FUNCTION_BLOCK UR (* Tamplate for a simple Basic Function Block Type *)
  (* Standard: 61499-2 *)
  (* Version 0.0, 2018-01-18, 4DIAC-IDE, 4DIAC-Consortium *)
  (* Version 1.0, 2016-05-26, AZ, fortiss GmbH *)
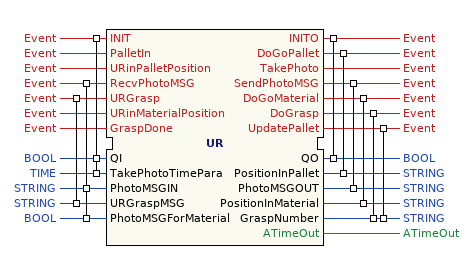
  EVENT_INPUT
    INIT WITH QI, TakePhotoTimePara; (* Initialization Request *)
    PalletIn; (* Normal Execution Request *)
    URinPalletPosition;
    RecvPhotoMSG WITH PhotoMSGIN, PhotoMSGForMaterial;
    URGrasp WITH URGraspMSG;
    URinMaterialPosition;
    GraspDone;
  END_EVENT
  EVENT_OUTPUT
    INITO WITH QO; (* Initialization Confirm *)
    DoGoPallet WITH PositionInPallet; (* send to real UR by socket *)
    TakePhoto; (* connnect to photo fb *)
    SendPhotoMSG WITH PhotoMSGOUT; (* send to pallet fb *)
    DoGoMaterial WITH PositionInMaterial;
    DoGrasp WITH GraspNumber;
    UpdatePallet WITH GraspNumber;
  END_EVENT
  VAR_INPUT
    QI : BOOL; (* Input event qualifier *)
    TakePhotoTimePara : TIME;
    PhotoMSGIN : STRING;
    URGraspMSG : STRING;
    PhotoMSGForMaterial : BOOL;
  END_VAR
  VAR_OUTPUT
    QO : BOOL; (* Output event qualifier *)
    PositionInPallet : STRING;
    PhotoMSGOUT : STRING;
    PositionInMaterial : STRING;
    GraspNumber : STRING;
  END_VAR
  PLUGS
    ATimeOut : ATimeOut;
  END_PLUGS
  VAR
    isFirst : BOOL; (* Is the first time to take photo， if true send 65 position to UR else send 66 *)
    isMSGForPallet : BOOL; (* If true, the MSG is for Pallet *)
  END_VAR
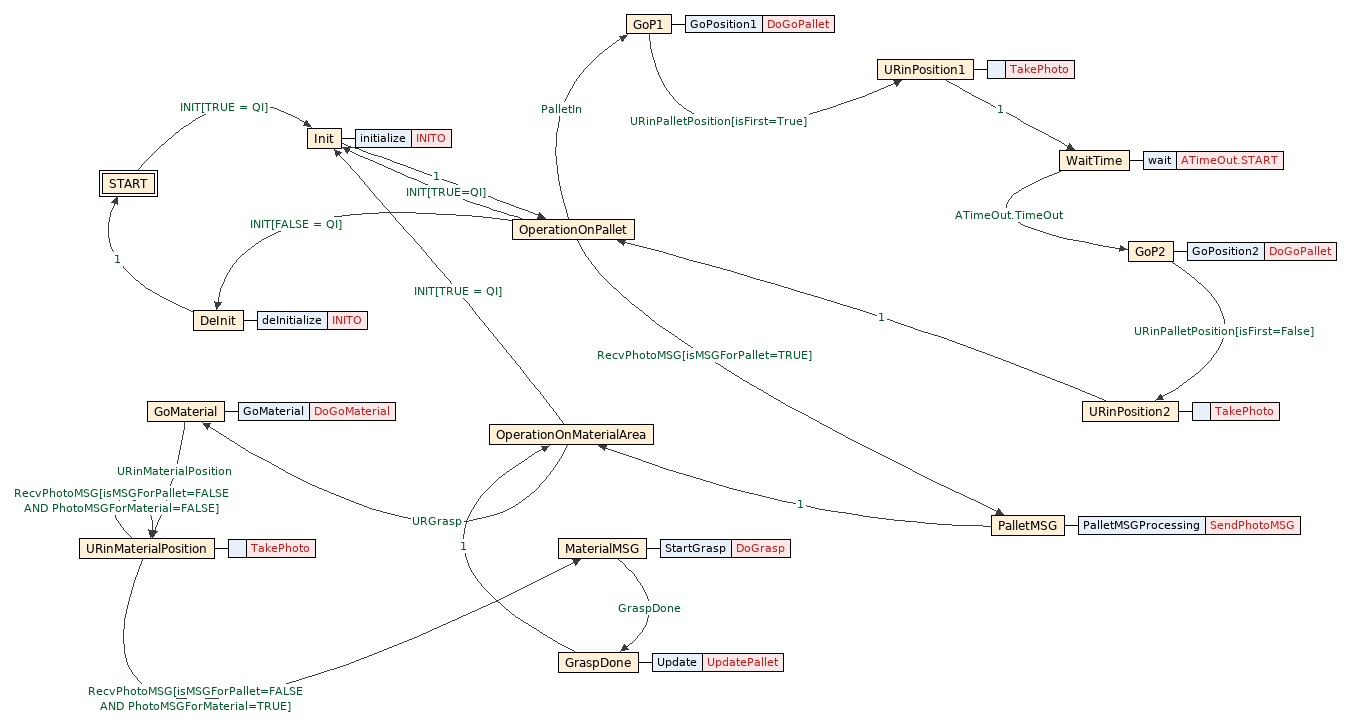
  EC_STATES
    START; (* Initial State *)
    Init : initialize -> INITO; (* Initialization *)
    GoP1 : GoPosition1 -> DoGoPallet; (* Normal execution *)
    OperationOnPallet;
    DeInit : deInitialize -> INITO;
    URinPosition1 : -> TakePhoto;
    WaitTime : wait -> ATimeOut.START;
    GoP2 : GoPosition2 -> DoGoPallet;
    URinPosition2 : -> TakePhoto;
    PalletMSG : PalletMSGProcessing -> SendPhotoMSG;
    MaterialMSG : StartGrasp -> DoGrasp;
    OperationOnMaterialArea;
    GoMaterial : GoMaterial -> DoGoMaterial;
    URinMaterialPosition : -> TakePhoto;
    GraspDone : Update -> UpdatePallet;
  END_STATES
  EC_TRANSITIONS
    START TO Init := INIT[TRUE = QI];
    Init TO OperationOnPallet := 1;
    OperationOnPallet TO GoP1 := PalletIn;
    DeInit TO START := 1;
    OperationOnPallet TO DeInit := INIT[FALSE = QI];
    OperationOnPallet TO PalletMSG := RecvPhotoMSG[isMSGForPallet=TRUE];
    GoP1 TO URinPosition1 := URinPalletPosition[isFirst=True];
    WaitTime TO GoP2 := ATimeOut.TimeOut;
    GoP2 TO URinPosition2 := URinPalletPosition[isFirst=False];
    URinPosition2 TO OperationOnPallet := 1;
    PalletMSG TO OperationOnMaterialArea := 1;
    OperationOnMaterialArea TO GoMaterial := URGrasp;
    GoMaterial TO URinMaterialPosition := URinMaterialPosition;
    URinMaterialPosition TO MaterialMSG := RecvPhotoMSG[isMSGForPallet=FALSE AND PhotoMSGForMaterial=TRUE];
    URinMaterialPosition TO URinMaterialPosition := RecvPhotoMSG[isMSGForPallet=FALSE AND PhotoMSGForMaterial=FALSE];
    MaterialMSG TO GraspDone := GraspDone;
    GraspDone TO OperationOnMaterialArea := 1;
    URinPosition1 TO WaitTime := 1;
    OperationOnMaterialArea TO Init := INIT[TRUE = QI];
    OperationOnPallet TO Init := INIT[TRUE=QI];
  END_TRANSITIONS
  ALGORITHM initialize IN ST: (* Initialization algorithm *)
isFirst:=TRUE;
isMSGForPallet:=TRUE;
PhotoMSGForMaterial:=FALSE;
PositionInPallet:= 0;
QO := QI;
  END_ALGORITHM
  ALGORITHM deInitialize IN ST: (* Normally executed algorithm *)
QO := FALSE;
  END_ALGORITHM
  ALGORITHM normalOperation IN ST: (* new algorithm *)
QO := QI;

IF TRUE  = QI THEN
  (*  only perform normal operation of QI is true*)

END_IF;
  END_ALGORITHM
  ALGORITHM GoPosition1 IN ST: (* new algorithm *)
PositionInPallet:='65';
isFirst:=TRUE;
  END_ALGORITHM
  ALGORITHM wait IN ST: (* new algorithm *)
ATimeOut.DT:=TakePhotoTimePara;
  END_ALGORITHM
  ALGORITHM GoPosition2 IN ST: (* new algorithm *)
PositionInPallet:='66';
isFirst:=FALSE;
isMSGForPallet:=TRUE;
  END_ALGORITHM
  ALGORITHM PalletMSGProcessing IN ST: (* new algorithm *)
PhotoMSGOUT:=PhotoMSGIN;
  END_ALGORITHM
  ALGORITHM StartGrasp IN ST: (* new algorithm *)
GraspNumber:=URGraspMSG;
  END_ALGORITHM
  ALGORITHM GoMaterial IN ST: (* new algorithm *)
PositionInMaterial:=URGraspMSG;
isMSGForPallet:=FALSE;
  END_ALGORITHM
  ALGORITHM Update IN ST: (* new algorithm *)
PhotoMSGForMaterial:=FALSE;
GraspNumber:=URGraspMSG;
  END_ALGORITHM
END_FUNCTION_BLOCK
